// TIA Portal V17 export
// export: Created 2025-03-07T09:23:48.8622662Z, ExportSetting WithDefaults, DisplayName Totally Integrated Automation Portal, DisplayVersion V17 Update 8, DisplayName TIA Portal Openness, DisplayVersion V17 Update 8, DisplayName TIA Portal Version Control Interface, DisplayVersion V17, DisplayName SINAMICS Startdrive Advanced, DisplayVersion V17 SP2, DisplayName SINAMICS Startdrive G110M, G120, G120C, G120D, G120P, G115D, DisplayVersion V17 SP2, DisplayName SINAMICS Startdrive G130, G150, S120, S150, SINAMICS MV, S210, DisplayVersion V17 SP2, DisplayName STEP 7 Professional, DisplayVersion V17 Update 8, DisplayName SINUMERIK ONE STEP 7 Toolbox, DisplayVersion V17 Update 12, DisplayName SINUMERIK 840D sl STEP 7 Toolbox, DisplayVersion V17 Update 12, DisplayName STEP 7 Safety, DisplayVersion V17 Update 6, DisplayName WinCC Advanced, DisplayVersion V17 Update 8
DATA_BLOCK "DB2040_WINCC_HMI_LINES"   // DB2040
{ S7_Optimized_Access := 'FALSE'; DB_Accessible_From_OPC_UA := 'FALSE' }
AUTHOR : ETXETAR
VERSION : 1.0
// stored: AutoNumber false, DBAccessibleFromOPCUA false, DBAccessibleFromWebserver true, IsOnlyStoredInLoadMemory false, IsWriteProtectedInAS false
   VAR RETAIN
      MODES { S7_SetPoint := 'True'} : Array[1..5] of "WINCC_HMI_LINES";
      SERVICES { S7_SetPoint := 'True'} : Array[1..30] of "WINCC_HMI_LINES";
   END_VAR
BEGIN
   // MODES[1] : AUTOMATIC MODE
   // MODES[2] : SEMIAUTO MODE
   // MODES[3] : MANUAL MODE
   // MODES[1].WINCC_LINE_REQUEST_RIGHT : AUTOMATIC MODE RIGHT REQUEST
   // MODES[2].WINCC_LINE_REQUEST_RIGHT : SEMIAUTO MODE RIGHT REQUEST
   // MODES[3].WINCC_LINE_REQUEST_RIGHT : MANUAL MODE RIGHT REQUEST
   // MODES[1].WINCC_LINE_REQUEST_LEFT : AUTOMATIC MODE LEFT REQUEST
   // MODES[2].WINCC_LINE_REQUEST_LEFT : SEMIAUTO MODE LEFT REQUEST
   // MODES[3].WINCC_LINE_REQUEST_LEFT : MANUAL MODE LEFT REQUEST
   // MODES[1].WINCC_LINE_CONDITIONS_RIGHT : AUTOMATIC MODE RIGHT CONDITIONS
   // MODES[2].WINCC_LINE_CONDITIONS_RIGHT : SEMIAUTO MODE RIGHT CONDITIONS
   // MODES[3].WINCC_LINE_CONDITIONS_RIGHT : MANUAL MODE RIGHT CONDITIONS
   // MODES[1].WINCC_LINE_CONDITIONS_LEFT : AUTOMATIC MODE LEFT CONDITIONS
   // MODES[2].WINCC_LINE_CONDITIONS_LEFT : SEMIAUTO MODE LEFT CONDITIONS
   // MODES[3].WINCC_LINE_CONDITIONS_LEFT : MANUAL MODE LEFT CONDITIONS
   // MODES[1].WINCC_LINE_ACTIVE_RIGHT : AUTOMATIC MODE RIGHT ACTIVE
   // MODES[2].WINCC_LINE_ACTIVE_RIGHT : SEMIAUTO MODE RIGHT ACTIVE
   // MODES[3].WINCC_LINE_ACTIVE_RIGHT : MANUAL MODE RIGHT ACTIVE
   // MODES[1].WINCC_LINE_ACTIVE_LEFT : AUTOMATIC MODE LEFT ACTIVE
   // MODES[2].WINCC_LINE_ACTIVE_LEFT : SEMIAUTO MODE LEFT ACTIVE
   // MODES[3].WINCC_LINE_ACTIVE_LEFT : MANUAL MODE LEFT ACTIVE
   // MODES[1].WINCC_LINE_STATUS_1_RIGHT : AUTOMATIC MODE RIGHT STATUS
   // MODES[2].WINCC_LINE_STATUS_1_RIGHT : SEMIAUTO MODE RIGHT STATUS
   // MODES[3].WINCC_LINE_STATUS_1_RIGHT : MANUAL MODE RIGHT STATUS
   // MODES[1].WINCC_LINE_STATUS_1_LEFT : AUTOMATIC MODE LEFT STATUS
   // MODES[2].WINCC_LINE_STATUS_1_LEFT : SEMIAUTO MODE LEFT STATUS
   // MODES[3].WINCC_LINE_STATUS_1_LEFT : MANUAL MODE LEFT STATUS
   // SERVICES[1] : PNEUMATIC SYSTEM
   // SERVICES[2] : POWDER FEEDER 1 GENERAL UNIT 01
   // SERVICES[3] : POWDER FEEDER 1 GENERAL UNIT 02
   // SERVICES[4] : POWDER FEEDER 2 GENERAL UNIT 02
   // SERVICES[5] : POWDER FEEDER 1 HEATER JKL UNIT 01 LINE 1
   // SERVICES[6] : POWDER FEEDER 1 HEATER JKL UNIT 01 LINE 2
   // SERVICES[7] : POWDER FEEDER 1 HEATER JKL UNIT 02 LINE 1
   // SERVICES[8] : POWDER FEEDER 1 HEATER JKL UNIT 02 LINE 2
   // SERVICES[9] : POWDER FEEDER 2 HEATER JKL UNIT 02 LINE 1
   // SERVICES[10] : POWDER FEEDER 1 HOPPER UNIT 01 LINE 1
   // SERVICES[11] : POWDER FEEDER 1 HOPPER UNIT 01 LINE 2
   // SERVICES[12] : POWDER FEEDER 1 HOPPER UNIT 02 LINE 1
   // SERVICES[13] : POWDER FEEDER 1 HOPPER UNIT 02 LINE 2
   // SERVICES[14] : POWDER FEEDER 2 HOPPER UNIT 02 LINE 1
END_DATA_BLOCK
